// Mitsubishi GX Works2 project: PLC_인터락   PLC: Q03UD

PROGRAM SHC
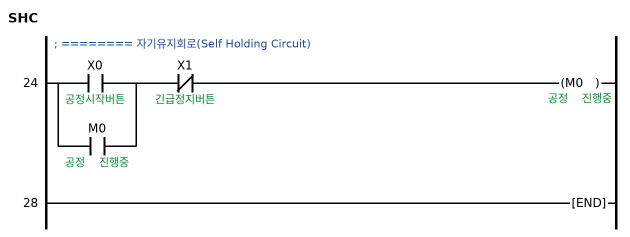
; ======== 자기유지회로(Self Holding Circuit)
24    LD      X0  ; 공정시작버튼
      OR      M0  ; 공정    진행중
      ANI     X1  ; 긴급정지버튼
      OUT     M0  ; 공정    진행중
28    END
END_PROGRAM

PROGRAM SetRst
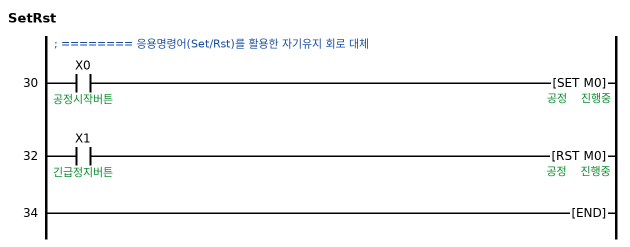
; ======== 응용명령어(Set/Rst)를 활용한 자기유지 회로 대체
30    LD      X0  ; 공정시작버튼
      SET     M0  ; 공정    진행중
32    LD      X1  ; 긴급정지버튼
      RST     M0  ; 공정    진행중
34    END
END_PROGRAM

PROGRAM IR
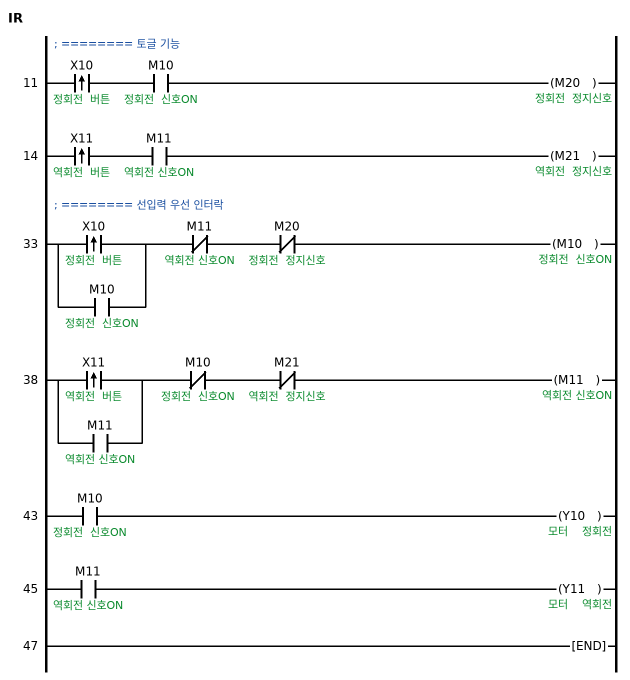
; ======== 토글 기능
11    LDP     X10  ; 정회전  버튼
      AND     M10  ; 정회전  신호ON
      OUT     M20  ; 정회전  정지신호
14    LDP     X11  ; 역회전  버튼
      AND     M11  ; 역회전 신호ON
      OUT     M21  ; 역회전  정지신호
; ======== 선입력 우선 인터락
33    LDP     X10  ; 정회전  버튼
      OR      M10  ; 정회전  신호ON
      ANI     M11  ; 역회전 신호ON
      ANI     M20  ; 정회전  정지신호
      OUT     M10  ; 정회전  신호ON
38    LDP     X11  ; 역회전  버튼
      OR      M11  ; 역회전 신호ON
      ANI     M10  ; 정회전  신호ON
      ANI     M21  ; 역회전  정지신호
      OUT     M11  ; 역회전 신호ON
43    LD      M10  ; 정회전  신호ON
      OUT     Y10  ; 모터    정회전
45    LD      M11  ; 역회전 신호ON
      OUT     Y11  ; 모터    역회전
47    END
END_PROGRAM

PROGRAM IRAfter
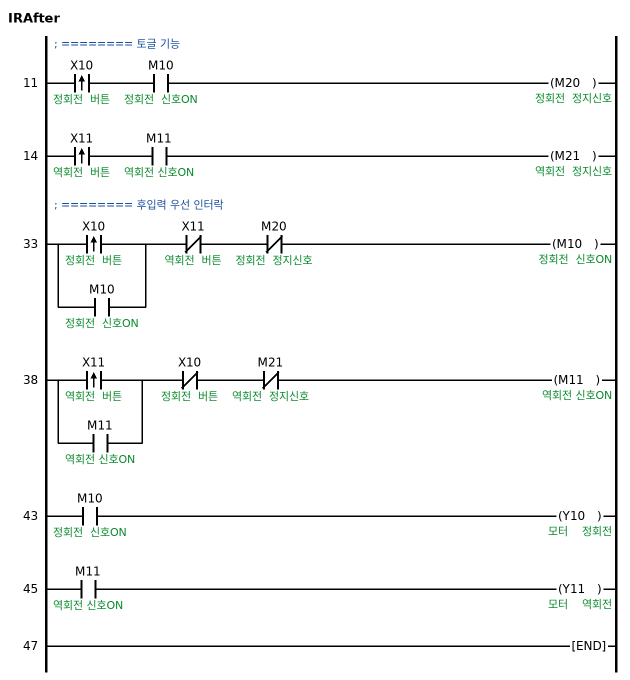
; ======== 토글 기능
11    LDP     X10  ; 정회전  버튼
      AND     M10  ; 정회전  신호ON
      OUT     M20  ; 정회전  정지신호
14    LDP     X11  ; 역회전  버튼
      AND     M11  ; 역회전 신호ON
      OUT     M21  ; 역회전  정지신호
; ======== 후입력 우선 인터락
33    LDP     X10  ; 정회전  버튼
      OR      M10  ; 정회전  신호ON
      ANI     X11  ; 역회전  버튼
      ANI     M20  ; 정회전  정지신호
      OUT     M10  ; 정회전  신호ON
38    LDP     X11  ; 역회전  버튼
      OR      M11  ; 역회전 신호ON
      ANI     X10  ; 정회전  버튼
      ANI     M21  ; 역회전  정지신호
      OUT     M11  ; 역회전 신호ON
43    LD      M10  ; 정회전  신호ON
      OUT     Y10  ; 모터    정회전
45    LD      M11  ; 역회전 신호ON
      OUT     Y11  ; 모터    역회전
47    END
END_PROGRAM

PROGRAM Invert
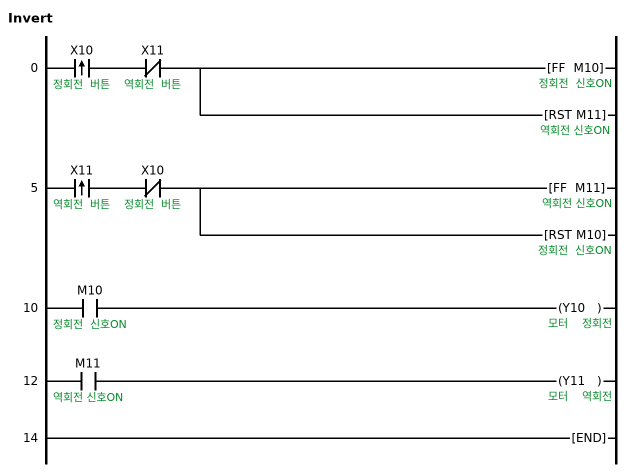
0     LDP     X10  ; 정회전  버튼
      ANI     X11  ; 역회전  버튼
      FF      M10  ; 정회전  신호ON
      RST     M11  ; 역회전 신호ON
5     LDP     X11  ; 역회전  버튼
      ANI     X10  ; 정회전  버튼
      FF      M11
      RST     M10  ; 정회전  신호ON
10    LD      M10  ; 정회전  신호ON
      OUT     Y10  ; 모터    정회전
12    LD      M11  ; 역회전 신호ON
      OUT     Y11  ; 모터    역회전
14    END
END_PROGRAM

// device comments not shown above
X3  ; PB3
